# EPICS substitutions: AFG3XXXSup/devAFG3XXX.substitutions
file "devAFG3XXXheader.template" {
    pattern { P, PORT }
	{ "\$(P)", "\$(PORT)" }
}

file "devAFG3XXXchannel.template" {
    pattern { P, PORT, C }
	{ "\$(P)", "\$(PORT)", "1" }
	{ "\$(P)", "\$(PORT)", "2" }
}
